(* Schneider Machine Expert - Basic project A9 Set - Reset, file version 2.7.0.0 *)
(* ProjectInformations: Name=Novo projeto *)

HARDWARE
  Cpu 0: TM221M16R/G
  EthernetConfiguration: NetworkName=M221, IpAllocationMode=FixedAddress, IpAddress=0.0.0.0, SubnetMask=0.0.0.0
  SerialLineConfiguration: Baud=Baud19200, Parity=ParityEven, DataBits=DataBits8, StopBits=StopBits1, PhysicalMedium=PhysicalMediumRs485, TransmissionMode=TransmissionModeModbusRtu, SlaveId=1, Addressing=SlaveAddressing
  MastTask: UsePeriodScanMode=false, PeriodScan=100
  FastTask: Period=255
  CpuBehavior: StartingMode=StartAsPreviousState, AutoSaveRamOnEeprom=true, WatchdogPeriod=250

SYMBOLS  (address, symbol, comment, settings)

POU Novo POU
  (* SectionNumber=1 *)

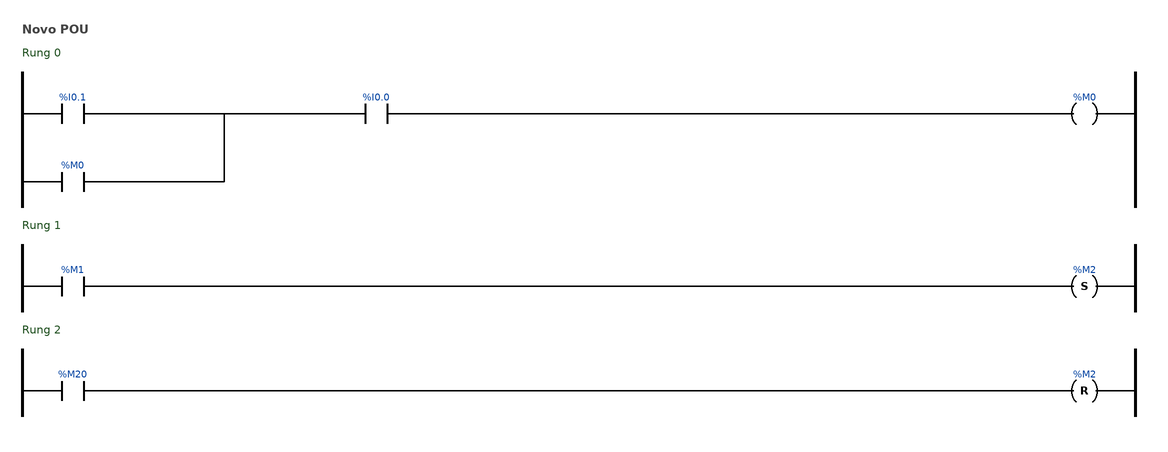

// Rung 0
  LD %I0.1
  OR %M0
  AND %I0.0
  ST %M0
  // as ST:
  //   %M0 := (%I0.1 OR %M0) AND %I0.0;

// Rung 1
  LD %M1
  S %M2
  // as ST:
  //   IF %M1 THEN %M2 := TRUE; END_IF;

// Rung 2
  LD %M20
  R %M2
  // as ST:
  //   IF %M20 THEN %M2 := FALSE; END_IF;
